VAR_GLOBAL
	instZufuehrbConveyorbelt	:	FactoryIO.FB_Foerderband;
	instAbholbConveyor	:	FactoryIO.FB_Foerderband;
	zufuehrbRunControlForwardActiv	:	BOOL;	//Runcontrol forward activ
	abholbRunControlForwardActiv	:	BOOL;	//Runcontrol forward activ
	instRunControl	:	FB_RunControl;
	simuActivateRunControl	:	BOOL;
	simuDeactivateRunControl	:	BOOL;
	simuRunControlActive	:	BOOL;
END_VAR

(* stored: Version 1.1.0.1
   GVL Conveyorbelts: Id {a16d026c-a3be-4f2b-bb6a-6cad3c9cf32b} *)
